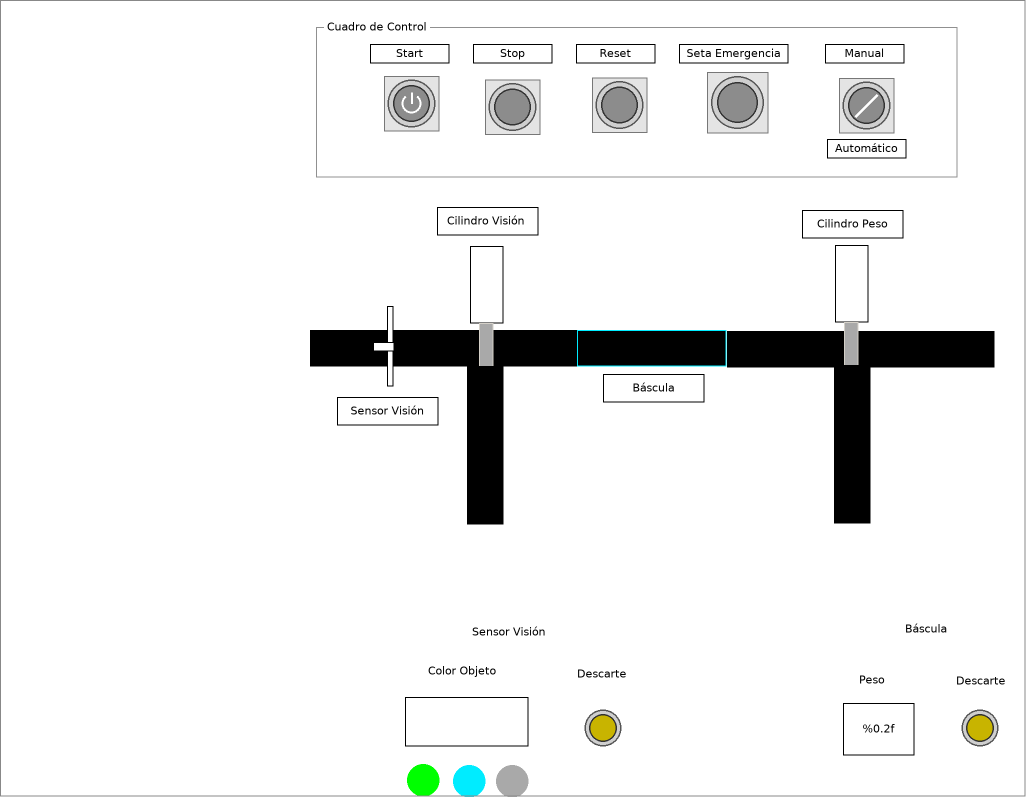
VISUALIZATION HMI  // 1026x797
    Label (430,605 158x54), "Sensor Visión"
    Lamp1 (582,704 42x48), variable: MAIN.descarteXcolor, style: Lamp-Lamp1-Yellow
    Label (557,659 90x30), "Descarte"
    Label (417,656 90x30), "Color Objeto"
    Label (847,602 158x54), "Báscula"
    Label (819,658 106x44), "Peso"
    Lamp1 (959,704 42x48), variable: MAIN.descratandoXpeso, style: Lamp-Lamp1-Yellow
    Label (936,666 90x30), "Descarte"
    Rectangle (405,697 123x49), text list: 'coloresSensorVision', text index: GVLvars.sVision
    Ellipse (407,764 32x32), invisible if: not Main.verde
    Ellipse (453,765 32x32), invisible if: not MAIN.azul
    Ellipse (496,765 32x32), colour toggle: MAIN.metal, invisible if: not MAIN.metal
    Rectangle (843,703 71x52), "%0.2f", text variable: MAIN.peso
    GroupBox (316,19 641x158), "Cuadro de Control"
        PowerSwitch (64,57 63x55), variable: GVLvars.botonStart, behaviour: TOGGLE, style: Switch-PowerSwitch-Gray
        PushSwitch (169,58 55x60), variable: GVLvars.botonStop, behaviour: TOGGLE, style: Switch-PushSwitch-Gray
        PushSwitch (276,56 55x60), variable: GVLvars.botonReset, behaviour: TOGGLE, style: Switch-PushSwitch-Gray
        PushSwitchLed (390,53 63x61), variable: GVLvars.setaEmergencia, behaviour: TOGGLE, style: Switch-PushSwitchLed-Gray
        Rectangle (54,25 79x19), "Start"
        Rectangle (157,25 79x19), "Stop"
        Rectangle (260,25 79x19), "Reset"
        Rectangle (363,25 109x19), "Seta Emergencia"
        Rectangle (509,25 79x19), "Manual"
        Rectangle (511,120 79x19), "Automático"
        RotarySwitch (523,59 55x55), variable: GVLvars.modoManual, behaviour: TOGGLE, style: Switch-RotarySwitch-Gray
    Rectangle (310,330 267x36), colour toggle: GVLvars.cintaVision
        toggle GVLvars.cintaVision
    Rectangle (727,331 267x36)
        toggle GVLvars.cintaPostBascula
    Rectangle (577,330 149x36), colour toggle: GVLvars.cintaBascula
        toggle GVLvars.cintaBascula
    Rectangle (470,246 33x77)
    Rectangle (479,323 14x77), invisible if: NOT GVLvars.cilindroVision
    Rectangle (437,207 101x28), "Cilindro Visión"
    Rectangle (835,245 33x77)
    Rectangle (844,322 14x77), invisible if: NOT GVLvars.cilindroBascula
    Rectangle (802,210 101x28), "Cilindro Peso"
    Rectangle (406,427 158x36), angle 90, colour toggle: GVLvars.cintaRemoveVision
        toggle GVLvars.cintaRemoveVision
    Rectangle (773,426 158x36), angle 90
        toggle GVLvars.cintaRemoveBascula
    Rectangle (603,374 101x28), "Báscula"
    Rectangle (350,343 80x6), angle 90
    Rectangle (373,342 21x9), angle 89
    Rectangle (337,397 101x28), "Sensor Visión"
END_VISUALIZATION

(* stored: Version 1.1.0.1, ProductVersion 3.1.4024.15
   Visu HMI: Id {a4cc15d2-b7c0-40f3-ac85-8780026a7f5f} *)
